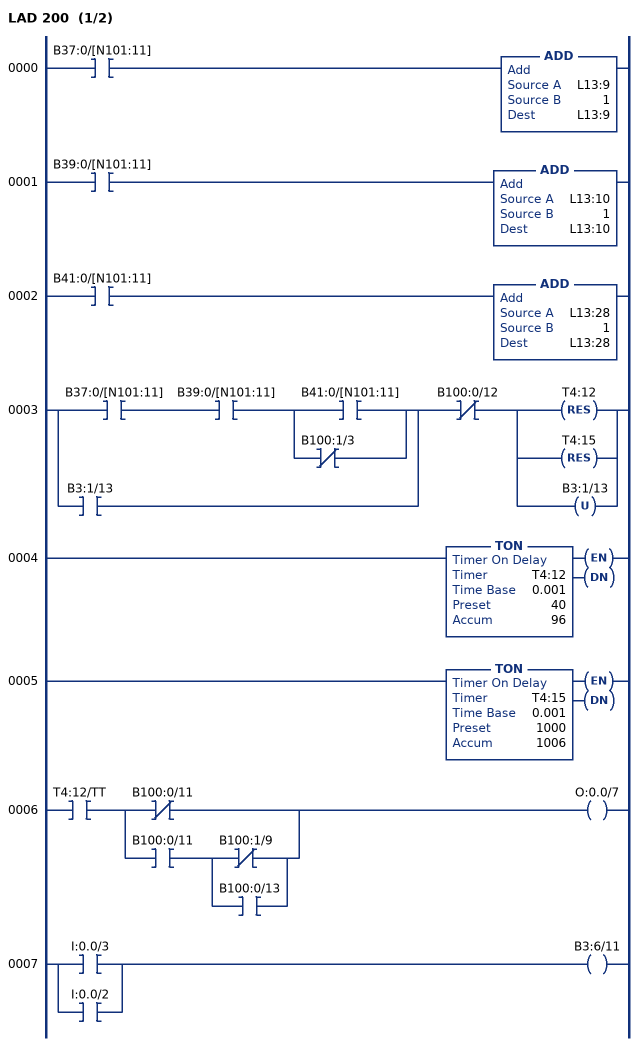
% Rung: 0 %
SOR XIC B37:0/[N101:11] ADD L13:9 1 L13:9 EOR
% Rung: 1 %
SOR XIC B39:0/[N101:11] ADD L13:10 1 L13:10 EOR
% Rung: 2 %
SOR XIC B41:0/[N101:11] ADD L13:28 1 L13:28 EOR
% Rung: 3 %
SOR BST XIC B37:0/[N101:11] XIC B39:0/[N101:11] BST XIC B41:0/[N101:11] NXB XIO B100:1/3 BND NXB XIC B3:1/13 BND XIO B100:0/12 BST RES T4:12 NXB RES T4:15 NXB OTU B3:1/13 BND EOR
% Rung: 4 %
SOR TON T4:12 0.001 40 96 EOR
% Rung: 5 %
SOR TON T4:15 0.001 1000 1006 EOR
% Rung: 6 %
SOR XIC T4:12/TT BST XIO B100:0/11 NXB XIC B100:0/11 BST XIO B100:1/9 NXB XIC B100:0/13 BND BND OTE O:0.0/7 EOR
% Rung: 7 %
SOR BST XIC I:0.0/3 NXB XIC I:0.0/2 BND OTE B3:6/11 EOR

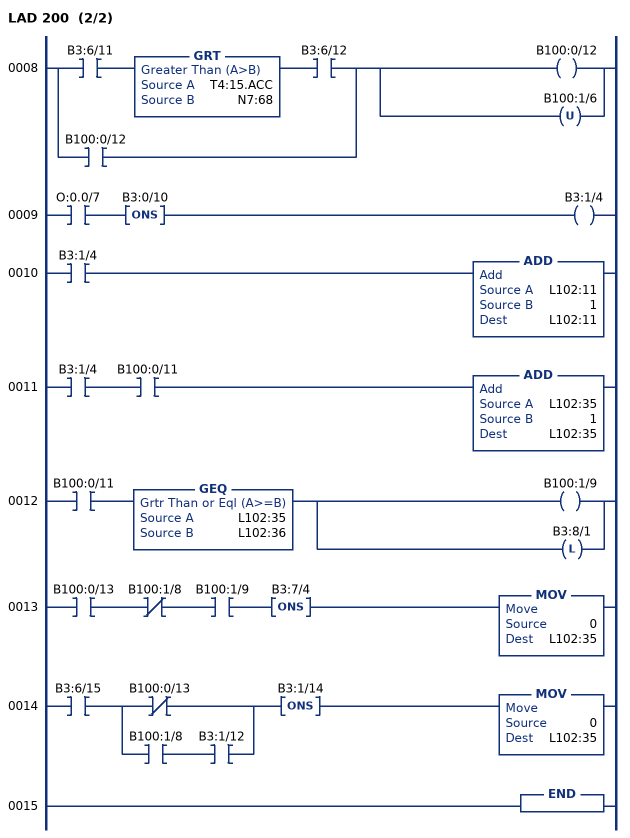
% Rung: 8 %
SOR BST XIC B3:6/11 GRT T4:15.ACC N7:68 XIC B3:6/12 NXB XIC B100:0/12 BND BST OTE B100:0/12 NXB OTU B100:1/6 BND EOR
% Rung: 9 %
SOR XIC O:0.0/7 ONS B3:0/10 OTE B3:1/4 EOR
% Rung: 10 %
SOR XIC B3:1/4 ADD L102:11 1 L102:11 EOR
% Rung: 11 %
SOR XIC B3:1/4 XIC B100:0/11 ADD L102:35 1 L102:35 EOR
% Rung: 12 %
SOR XIC B100:0/11 GEQ L102:35 L102:36 BST OTE B100:1/9 NXB OTL B3:8/1 BND EOR
% Rung: 13 %
SOR XIC B100:0/13 XIO B100:1/8 XIC B100:1/9 ONS B3:7/4 MOV 0 L102:35 EOR
% Rung: 14 %
SOR XIC B3:6/15 BST XIO B100:0/13 NXB XIC B100:1/8 XIC B3:1/12 BND ONS B3:1/14 MOV 0 L102:35 EOR
% Rung: 15 %
SOR END EOR

LADDER 235
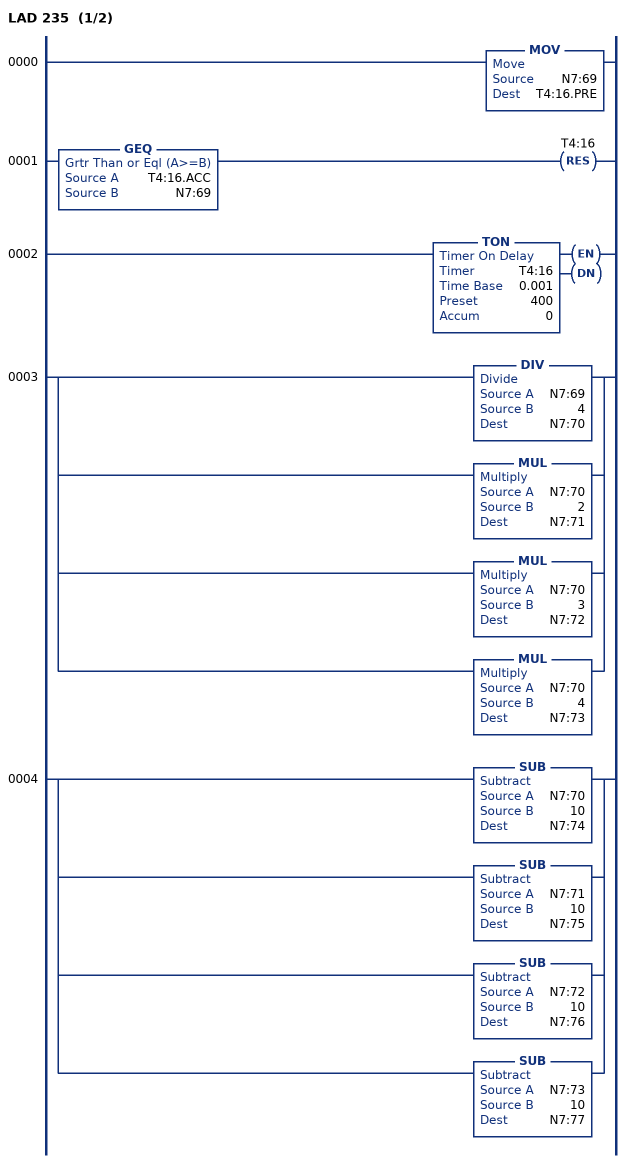
% Rung: 0 %
SOR MOV N7:69 T4:16.PRE EOR
% Rung: 1 %
SOR GEQ T4:16.ACC N7:69 RES T4:16 EOR
% Rung: 2 %
SOR TON T4:16 0.001 400 0 EOR
% Rung: 3 %
SOR BST DIV N7:69 4 N7:70 NXB MUL N7:70 2 N7:71 NXB MUL N7:70 3 N7:72 NXB MUL N7:70 4 N7:73 BND EOR
% Rung: 4 %
SOR BST SUB N7:70 10 N7:74 NXB SUB N7:71 10 N7:75 NXB SUB N7:72 10 N7:76 NXB SUB N7:73 10 N7:77 BND EOR

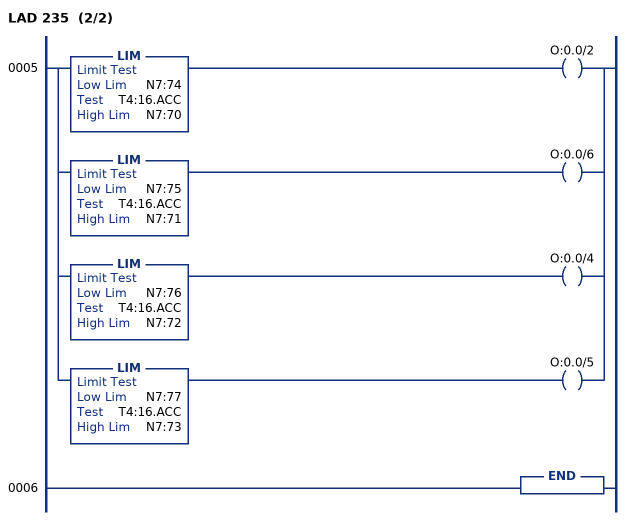
% Rung: 5 %
SOR BST LIM N7:74 T4:16.ACC N7:70 OTE O:0.0/2 NXB LIM N7:75 T4:16.ACC N7:71 OTE O:0.0/6 NXB LIM N7:76 T4:16.ACC N7:72 OTE O:0.0/4 NXB LIM N7:77 T4:16.ACC N7:73 OTE O:0.0/5 BND EOR
% Rung: 6 %
SOR END EOR

LADDER 236
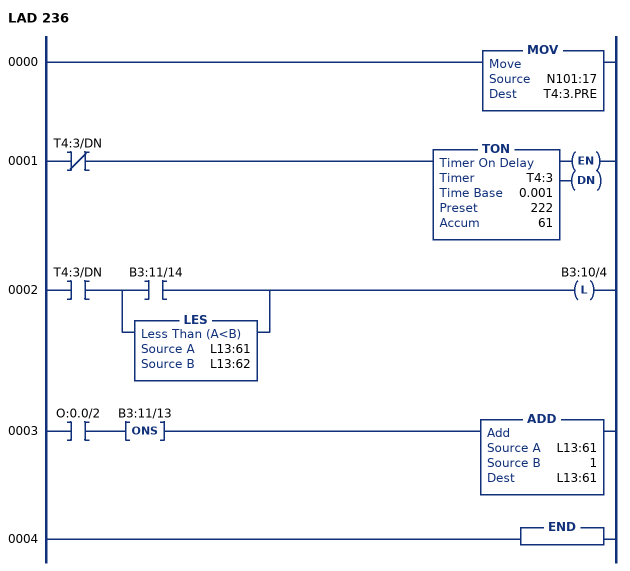
% Rung: 0 %
SOR MOV N101:17 T4:3.PRE EOR
% Rung: 1 %
SOR XIO T4:3/DN TON T4:3 0.001 222 61 EOR
% Rung: 2 %
SOR XIC T4:3/DN BST XIC B3:11/14 NXB LES L13:61 L13:62 BND OTL B3:10/4 EOR
% Rung: 3 %
SOR XIC O:0.0/2 ONS B3:11/13 ADD L13:61 1 L13:61 EOR
% Rung: 4 %
SOR END EOR

LADDER 237
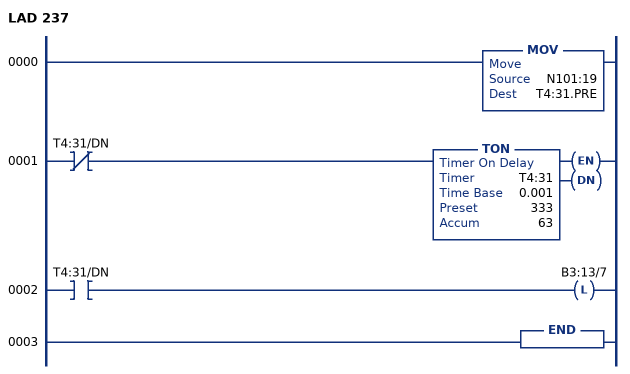
% Rung: 0 %
SOR MOV N101:19 T4:31.PRE EOR
% Rung: 1 %
SOR XIO T4:31/DN TON T4:31 0.001 333 63 EOR
% Rung: 2 %
SOR XIC T4:31/DN OTL B3:13/7 EOR
% Rung: 3 %
SOR END EOR

LADDER 238
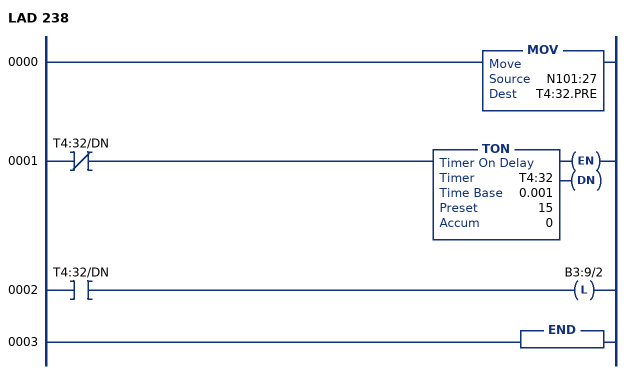
% Rung: 0 %
SOR MOV N101:27 T4:32.PRE EOR
% Rung: 1 %
SOR XIO T4:32/DN TON T4:32 0.001 15 0 EOR
% Rung: 2 %
SOR XIC T4:32/DN OTL B3:9/2 EOR
% Rung: 3 %
SOR END EOR

LADDER 239
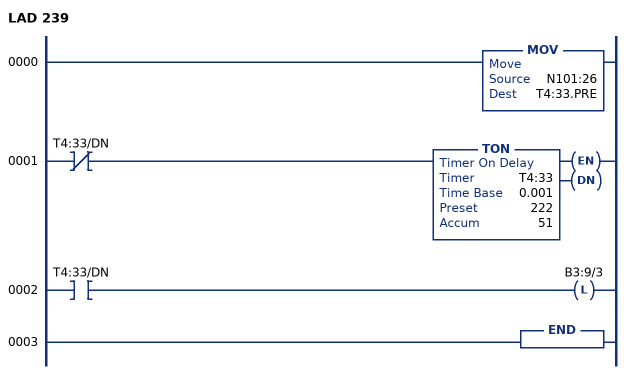
% Rung: 0 %
SOR MOV N101:26 T4:33.PRE EOR
% Rung: 1 %
SOR XIO T4:33/DN TON T4:33 0.001 222 51 EOR
% Rung: 2 %
SOR XIC T4:33/DN OTL B3:9/3 EOR
% Rung: 3 %
SOR END EOR

LADDER 240
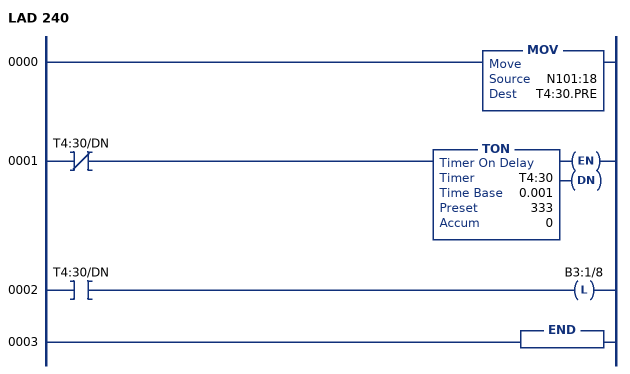
% Rung: 0 %
SOR MOV N101:18 T4:30.PRE EOR
% Rung: 1 %
SOR XIO T4:30/DN TON T4:30 0.001 333 0 EOR
% Rung: 2 %
SOR XIC T4:30/DN OTL B3:1/8 EOR
% Rung: 3 %
SOR END EOR

LADDER 241
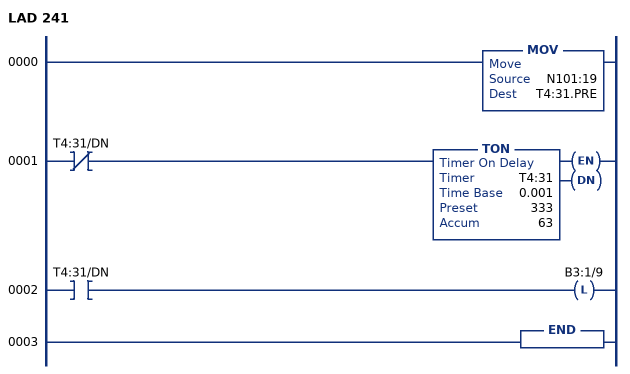
% Rung: 0 %
SOR MOV N101:19 T4:31.PRE EOR
% Rung: 1 %
SOR XIO T4:31/DN TON T4:31 0.001 333 63 EOR
% Rung: 2 %
SOR XIC T4:31/DN OTL B3:1/9 EOR
% Rung: 3 %
SOR END EOR

LADDER 242
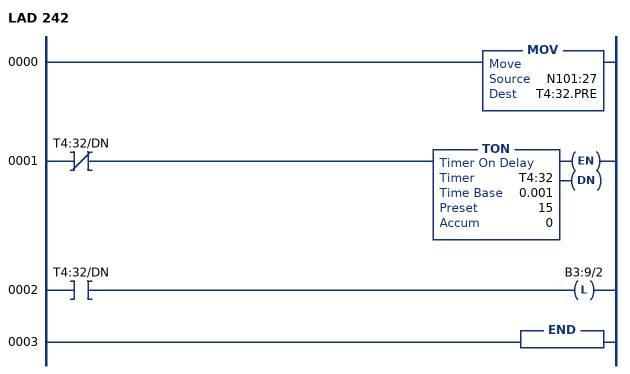
% Rung: 0 %
SOR MOV N101:27 T4:32.PRE EOR
% Rung: 1 %
SOR XIO T4:32/DN TON T4:32 0.001 15 0 EOR
% Rung: 2 %
SOR XIC T4:32/DN OTL B3:9/2 EOR
% Rung: 3 %
SOR END EOR

LADDER 243
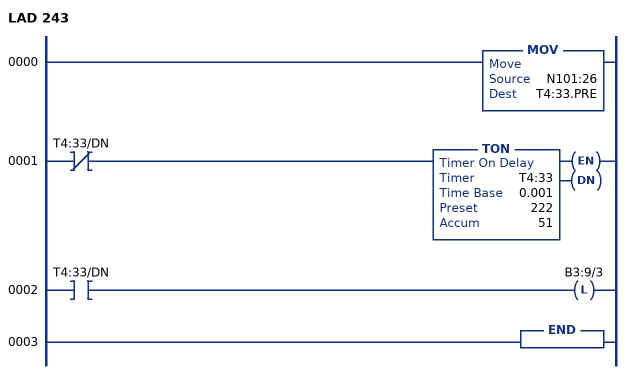
% Rung: 0 %
SOR MOV N101:26 T4:33.PRE EOR
% Rung: 1 %
SOR XIO T4:33/DN TON T4:33 0.001 222 51 EOR
% Rung: 2 %
SOR XIC T4:33/DN OTL B3:9/3 EOR
% Rung: 3 %
SOR END EOR

LADDER 244
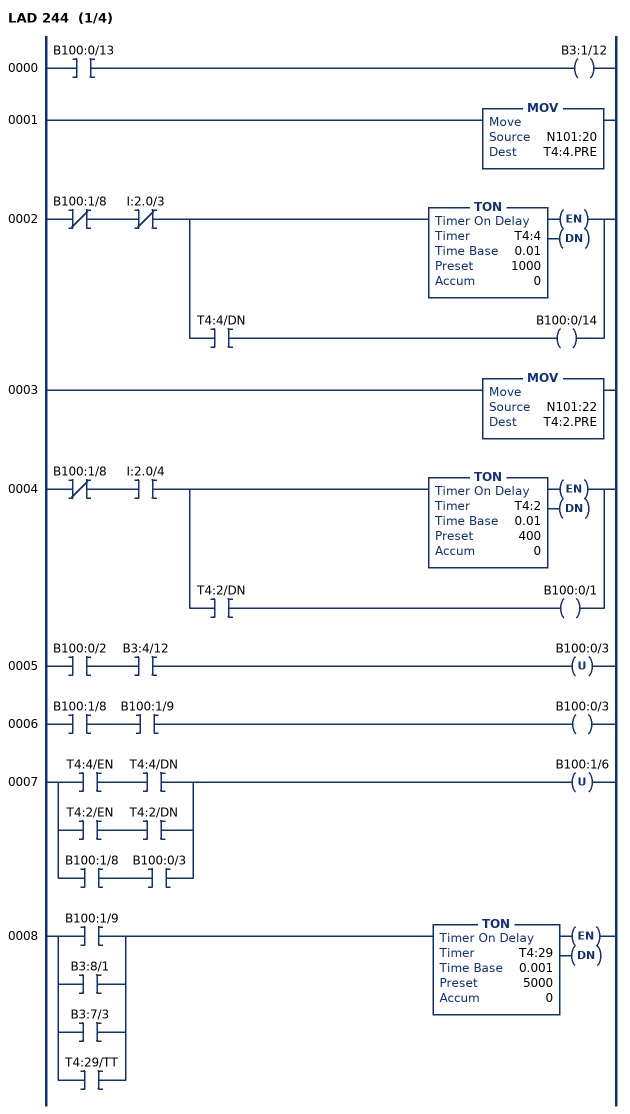
% Rung: 0 %
SOR XIC B100:0/13 OTE B3:1/12 EOR
% Rung: 1 %
SOR MOV N101:20 T4:4.PRE EOR
% Rung: 2 %
SOR XIO B100:1/8 XIO I:2.0/3 BST TON T4:4 0.01 1000 0 NXB XIC T4:4/DN OTE B100:0/14 BND EOR
% Rung: 3 %
SOR MOV N101:22 T4:2.PRE EOR
% Rung: 4 %
SOR XIO B100:1/8 XIC I:2.0/4 BST TON T4:2 0.01 400 0 NXB XIC T4:2/DN OTE B100:0/1 BND EOR
% Rung: 5 %
SOR XIC B100:0/2 XIC B3:4/12 OTU B100:0/3 EOR
% Rung: 6 %
SOR XIC B100:1/8 XIC B100:1/9 OTE B100:0/3 EOR
% Rung: 7 %
SOR BST XIC T4:4/EN XIC T4:4/DN NXB XIC T4:2/EN XIC T4:2/DN NXB XIC B100:1/8 XIC B100:0/3 BND OTU B100:1/6 EOR
% Rung: 8 %
SOR BST XIC B100:1/9 NXB XIC B3:8/1 NXB XIC B3:7/3 NXB XIC T4:29/TT BND TON T4:29 0.001 5000 0 EOR

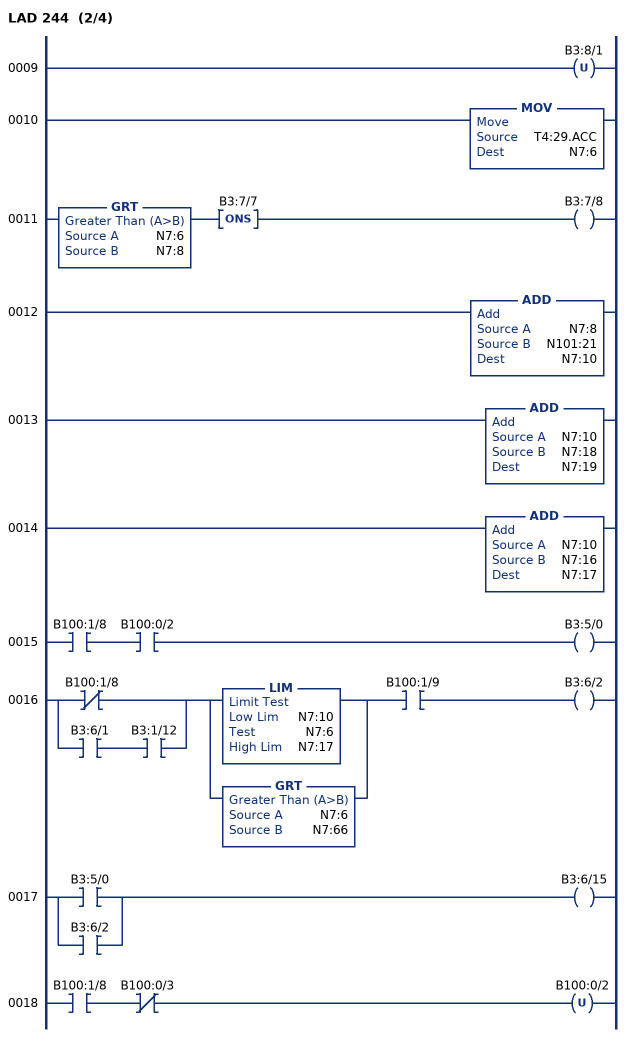
% Rung: 9 %
SOR OTU B3:8/1 EOR
% Rung: 10 %
SOR MOV T4:29.ACC N7:6 EOR
% Rung: 11 %
SOR GRT N7:6 N7:8 ONS B3:7/7 OTE B3:7/8 EOR
% Rung: 12 %
SOR ADD N7:8 N101:21 N7:10 EOR
% Rung: 13 %
SOR ADD N7:10 N7:18 N7:19 EOR
% Rung: 14 %
SOR ADD N7:10 N7:16 N7:17 EOR
% Rung: 15 %
SOR XIC B100:1/8 XIC B100:0/2 OTE B3:5/0 EOR
% Rung: 16 %
SOR BST XIO B100:1/8 NXB XIC B3:6/1 XIC B3:1/12 BND BST LIM N7:10 N7:6 N7:17 NXB GRT N7:6 N7:66 BND XIC B100:1/9 OTE B3:6/2 EOR
% Rung: 17 %
SOR BST XIC B3:5/0 NXB XIC B3:6/2 BND OTE B3:6/15 EOR
% Rung: 18 %
SOR XIC B100:1/8 XIO B100:0/3 OTU B100:0/2 EOR

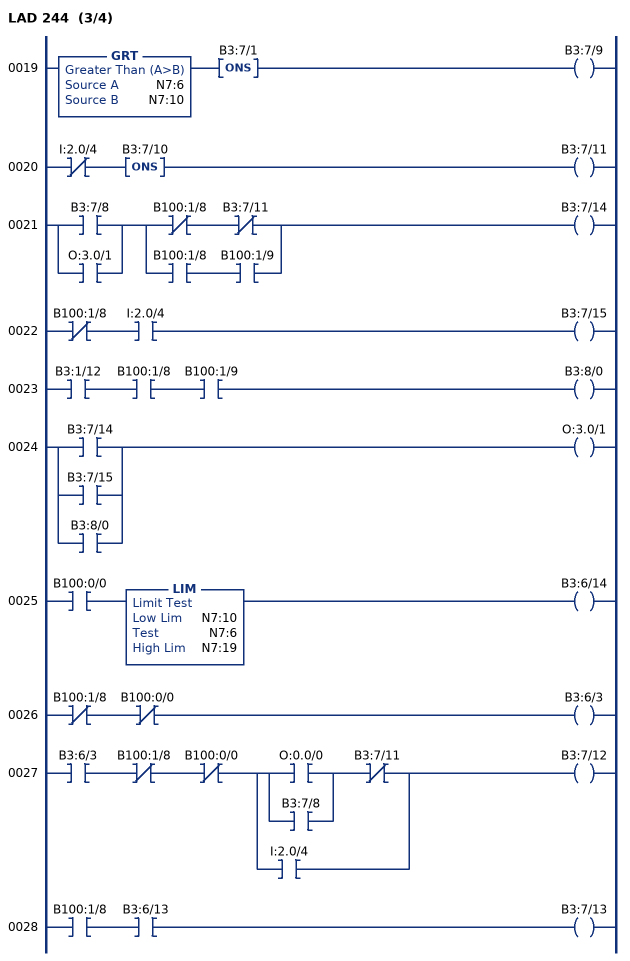
% Rung: 19 %
SOR GRT N7:6 N7:10 ONS B3:7/1 OTE B3:7/9 EOR
% Rung: 20 %
SOR XIO I:2.0/4 ONS B3:7/10 OTE B3:7/11 EOR
% Rung: 21 %
SOR BST XIC B3:7/8 NXB XIC O:3.0/1 BND BST XIO B100:1/8 XIO B3:7/11 NXB XIC B100:1/8 XIC B100:1/9 BND OTE B3:7/14 EOR
% Rung: 22 %
SOR XIO B100:1/8 XIC I:2.0/4 OTE B3:7/15 EOR
% Rung: 23 %
SOR XIC B3:1/12 XIC B100:1/8 XIC B100:1/9 OTE B3:8/0 EOR
% Rung: 24 %
SOR BST XIC B3:7/14 NXB XIC B3:7/15 NXB XIC B3:8/0 BND OTE O:3.0/1 EOR
% Rung: 25 %
SOR XIC B100:0/0 LIM N7:10 N7:6 N7:19 OTE B3:6/14 EOR
% Rung: 26 %
SOR XIO B100:1/8 XIO B100:0/0 OTE B3:6/3 EOR
% Rung: 27 %
SOR XIC B3:6/3 XIO B100:1/8 XIO B100:0/0 BST BST XIC O:0.0/0 NXB XIC B3:7/8 BND XIO B3:7/11 NXB XIC I:2.0/4 BND OTE B3:7/12 EOR
% Rung: 28 %
SOR XIC B100:1/8 XIC B3:6/13 OTE B3:7/13 EOR

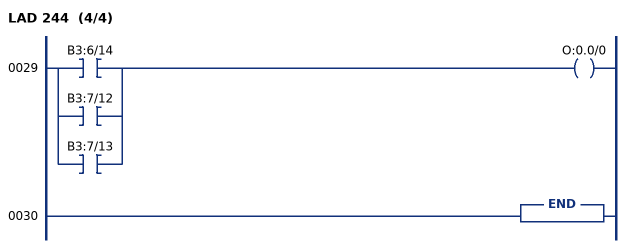
% Rung: 29 %
SOR BST XIC B3:6/14 NXB XIC B3:7/12 NXB XIC B3:7/13 BND OTE O:0.0/0 EOR
% Rung: 30 %
SOR END EOR

LADDER 245
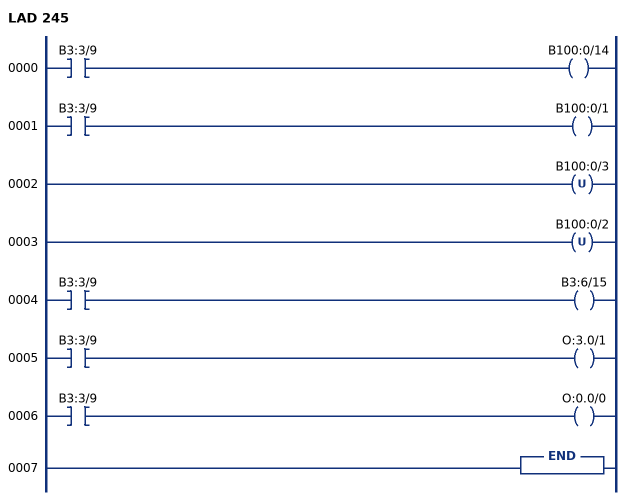
% Rung: 0 %
SOR XIC B3:3/9 OTE B100:0/14 EOR
% Rung: 1 %
SOR XIC B3:3/9 OTE B100:0/1 EOR
% Rung: 2 %
SOR OTU B100:0/3 EOR
% Rung: 3 %
SOR OTU B100:0/2 EOR
% Rung: 4 %
SOR XIC B3:3/9 OTE B3:6/15 EOR
% Rung: 5 %
SOR XIC B3:3/9 OTE O:3.0/1 EOR
% Rung: 6 %
SOR XIC B3:3/9 OTE O:0.0/0 EOR
% Rung: 7 %
SOR END EOR

LADDER 246
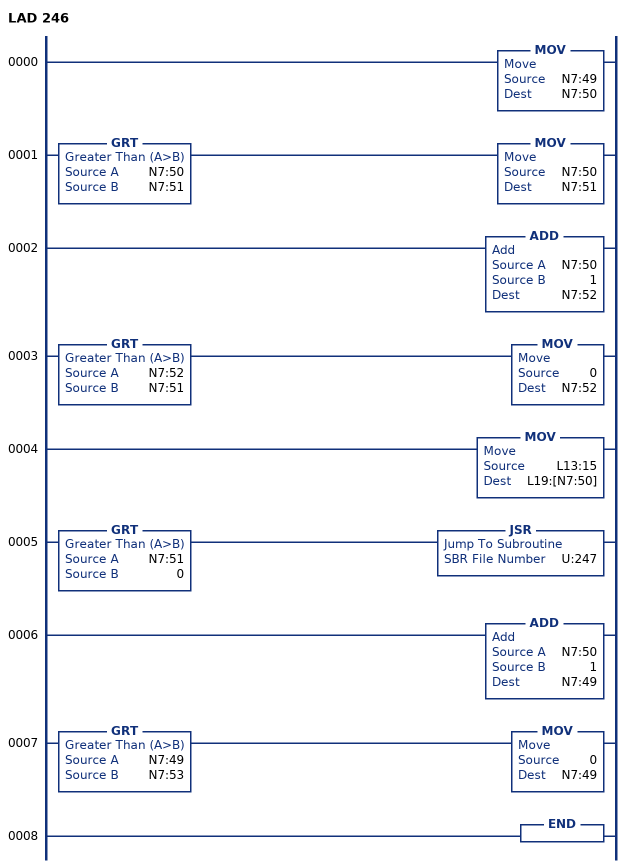
% Rung: 0 %
SOR MOV N7:49 N7:50 EOR
% Rung: 1 %
SOR GRT N7:50 N7:51 MOV N7:50 N7:51 EOR
% Rung: 2 %
SOR ADD N7:50 1 N7:52 EOR
% Rung: 3 %
SOR GRT N7:52 N7:51 MOV 0 N7:52 EOR
% Rung: 4 %
SOR MOV L13:15 L19:[N7:50] EOR
% Rung: 5 %
SOR GRT N7:51 0 JSR U:247 EOR
% Rung: 6 %
SOR ADD N7:50 1 N7:49 EOR
% Rung: 7 %
SOR GRT N7:49 N7:53 MOV 0 N7:49 EOR
% Rung: 8 %
SOR END EOR

LADDER 247
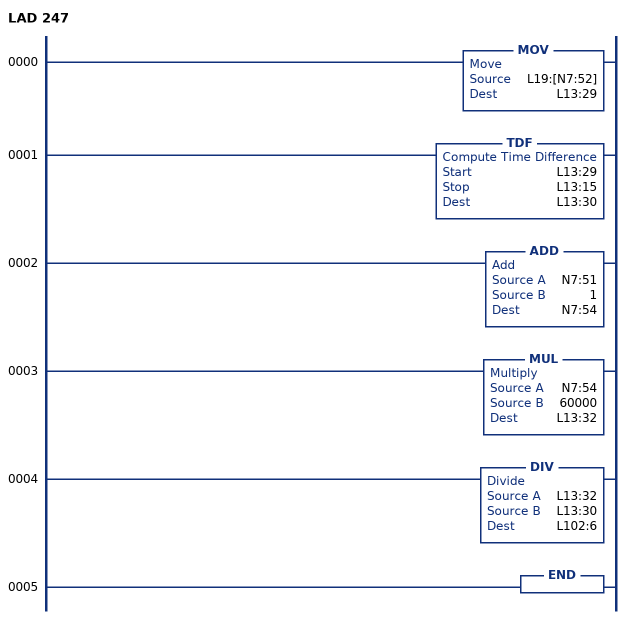
% Rung: 0 %
SOR MOV L19:[N7:52] L13:29 EOR
% Rung: 1 %
SOR TDF L13:29 L13:15 L13:30 EOR
% Rung: 2 %
SOR ADD N7:51 1 N7:54 EOR
% Rung: 3 %
SOR MUL N7:54 60000 L13:32 EOR
% Rung: 4 %
SOR DIV L13:32 L13:30 L102:6 EOR
% Rung: 5 %
SOR END EOR

LADDER 248
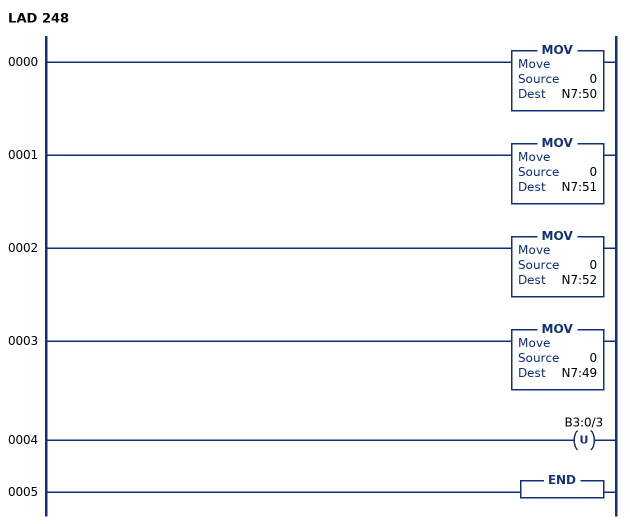
% Rung: 0 %
SOR MOV 0 N7:50 EOR
% Rung: 1 %
SOR MOV 0 N7:51 EOR
% Rung: 2 %
SOR MOV 0 N7:52 EOR
% Rung: 3 %
SOR MOV 0 N7:49 EOR
% Rung: 4 %
SOR OTU B3:0/3 EOR
% Rung: 5 %
SOR END EOR

LADDER 249
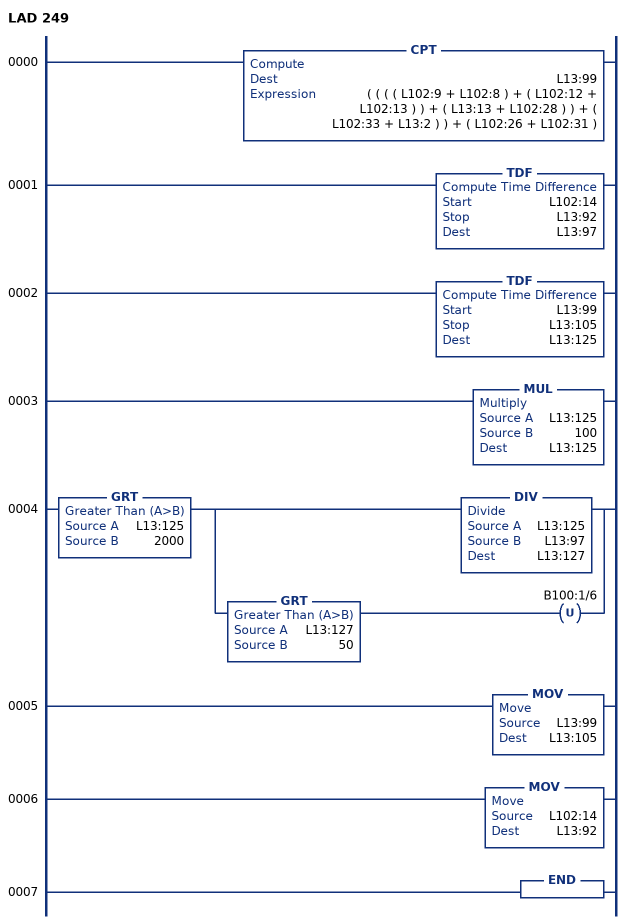
% Rung: 0 %
SOR CPT L13:99 " ( ( ( ( L102:9 + L102:8 ) + ( L102:12 + L102:13 ) ) + ( L13:13 + L102:28 ) ) + ( L102:33 + L13:2 ) ) + ( L102:26 + L102:31 ) " EOR
% Rung: 1 %
SOR TDF L102:14 L13:92 L13:97 EOR
% Rung: 2 %
SOR TDF L13:99 L13:105 L13:125 EOR
% Rung: 3 %
SOR MUL L13:125 100 L13:125 EOR
% Rung: 4 %
SOR GRT L13:125 2000 BST DIV L13:125 L13:97 L13:127 NXB GRT L13:127 50 OTU B100:1/6 BND EOR
% Rung: 5 %
SOR MOV L13:99 L13:105 EOR
% Rung: 6 %
SOR MOV L102:14 L13:92 EOR
% Rung: 7 %
SOR END EOR

LADDER 250
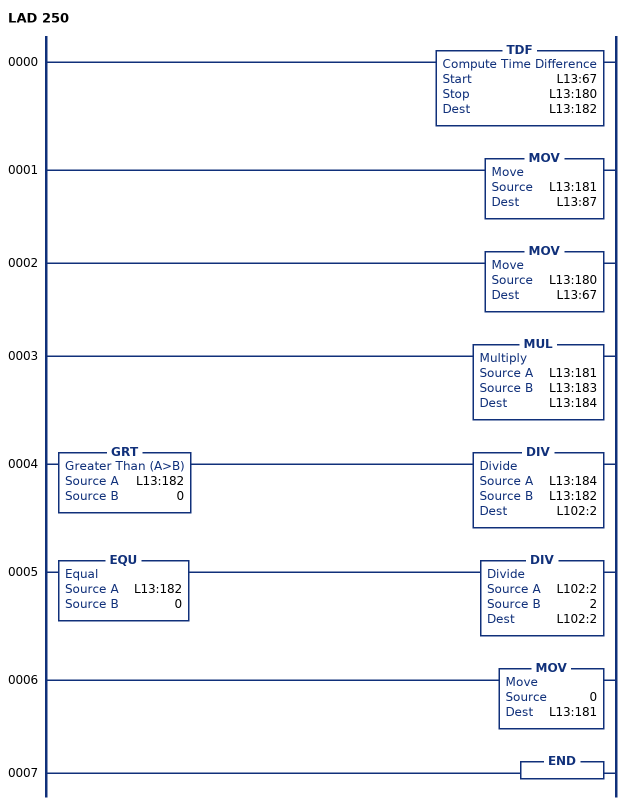
% Rung: 0 %
SOR TDF L13:67 L13:180 L13:182 EOR
% Rung: 1 %
SOR MOV L13:181 L13:87 EOR
% Rung: 2 %
SOR MOV L13:180 L13:67 EOR
% Rung: 3 %
SOR MUL L13:181 L13:183 L13:184 EOR
% Rung: 4 %
SOR GRT L13:182 0 DIV L13:184 L13:182 L102:2 EOR
% Rung: 5 %
SOR EQU L13:182 0 DIV L102:2 2 L102:2 EOR
% Rung: 6 %
SOR MOV 0 L13:181 EOR
% Rung: 7 %
SOR END EOR

LADDER 251
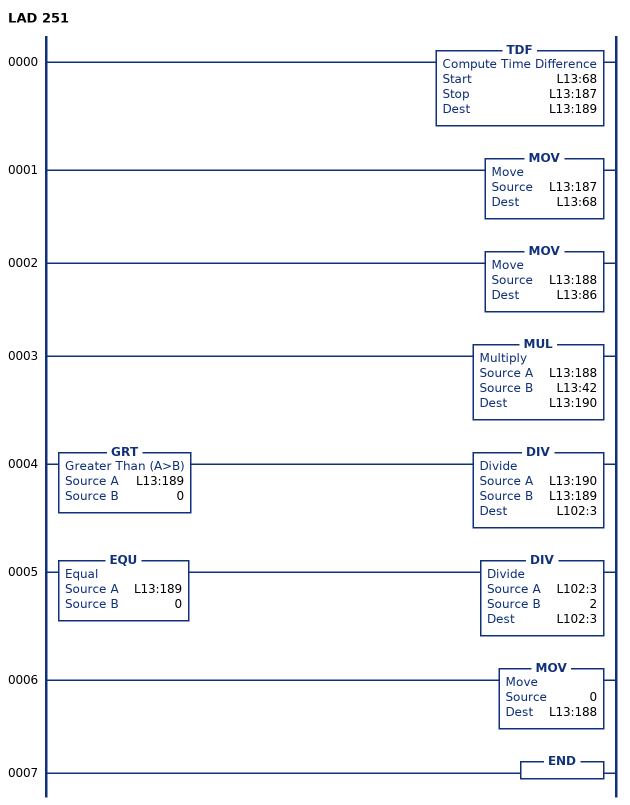
% Rung: 0 %
SOR TDF L13:68 L13:187 L13:189 EOR
% Rung: 1 %
SOR MOV L13:187 L13:68 EOR
% Rung: 2 %
SOR MOV L13:188 L13:86 EOR
% Rung: 3 %
SOR MUL L13:188 L13:42 L13:190 EOR
% Rung: 4 %
SOR GRT L13:189 0 DIV L13:190 L13:189 L102:3 EOR
% Rung: 5 %
SOR EQU L13:189 0 DIV L102:3 2 L102:3 EOR
% Rung: 6 %
SOR MOV 0 L13:188 EOR
% Rung: 7 %
SOR END EOR

LADDER 252
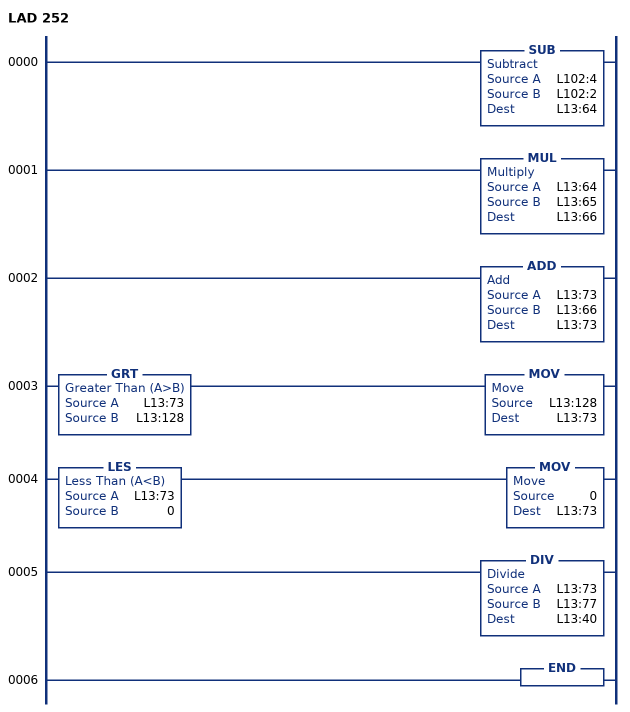
% Rung: 0 %
SOR SUB L102:4 L102:2 L13:64 EOR
% Rung: 1 %
SOR MUL L13:64 L13:65 L13:66 EOR
% Rung: 2 %
SOR ADD L13:73 L13:66 L13:73 EOR
% Rung: 3 %
SOR GRT L13:73 L13:128 MOV L13:128 L13:73 EOR
% Rung: 4 %
SOR LES L13:73 0 MOV 0 L13:73 EOR
% Rung: 5 %
SOR DIV L13:73 L13:77 L13:40 EOR
% Rung: 6 %
SOR END EOR

LADDER 253
